# EPICS autosave request: apps/scalerApp/Db/scaler16m_norm_settings.req
# FILE... scaler16m_norm_settings.req
# USAGE.. transform Record fields autosave'd.

file transform_settings.req P=$(P)_norm1
file transform_settings.req P=$(P)_norm2
